FUNCTION_BLOCK FB_HoneyFill IMPLEMENTS I_FillingStrategy

VAR
END_VAR

{warning 'add method implementation '}
METHOD ExecuteFill : BOOL
VAR_INPUT
	stBottle: REFERENCE TO ST_Bottle;
END_VAR
VAR CONSTANT
	cFILLING_SPEED : REAL := 2;
END_VAR
IF __ISVALIDREF(stBottle) THEN
	IF stBottle.fCurrentLevel >= stBottle.fTargetLevel THEN
		ExecuteFill := TRUE;
	ELSE
		stBottle.fCurrentLevel := stBottle.fCurrentLevel + cFILLING_SPEED;
		ExecuteFill := FALSE;
	END_IF
END_IF
END_METHOD

END_FUNCTION_BLOCK

(* stored: Version 1.1.0.1, ProductVersion 3.1.4024.16
   POU FB_HoneyFill: Id {bd95f233-1e19-4bbb-b629-4f43dd2f1f99}, SpecialFunc None
   Method ExecuteFill: Id {8dcba71c-4a5b-411a-b4f8-9259c9281d69} *)
